FUNCTION_BLOCK XCBR (* Composite Function Block Type *)
  (* Standard: 61499-2 *)
  (* Version 0.0, 12/11/2023, Cheyan, Schneider Electric, template *)
  PACKAGE Main;
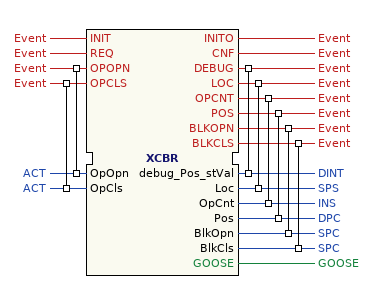
  EVENT_INPUT
    INIT; (* Initialization Request *)
    REQ; (* Normal Execution Request *)
    OPOPN WITH OpOpn;
    OPCLS WITH OpCls;
  END_EVENT
  EVENT_OUTPUT
    INITO; (* Initialization Confirm *)
    CNF; (* Execution Confirmation *)
    DEBUG WITH debug_Pos_stVal;
    LOC WITH Loc;
    OPCNT WITH OpCnt;
    POS WITH Pos;
    BLKOPN WITH BlkOpn;
    BLKCLS WITH BlkCls;
  END_EVENT
  VAR_INPUT
    OpOpn : ACT; (* Input event qualifier *)
    OpCls : ACT;
  END_VAR
  VAR_OUTPUT
    debug_Pos_stVal : DINT;
    Loc : SPS;
    OpCnt : INS;
    Pos : DPC;
    BlkOpn : SPC;
    BlkCls : SPC;
  END_VAR
  PLUGS
    GOOSE : GOOSE;
  END_PLUGS
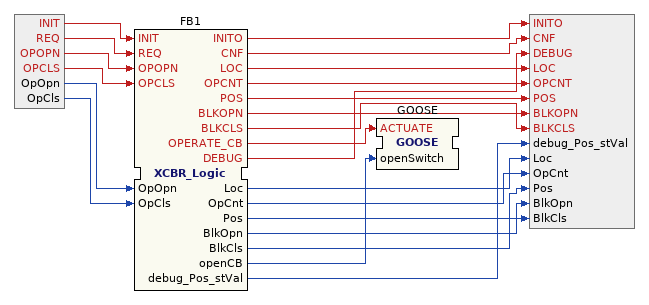
  FBS
    FB1 : XCBR_Logic;
  END_FBS
  EVENT_CONNECTIONS
    INIT TO FB1.INIT;
    REQ TO FB1.REQ;
    FB1.INITO TO INITO;
    FB1.CNF TO CNF;
    FB1.OPERATE_CB TO GOOSE.ACTUATE;
    FB1.DEBUG TO DEBUG;
    FB1.LOC TO LOC;
    FB1.OPCNT TO OPCNT;
    FB1.POS TO POS;
    FB1.BLKOPN TO BLKOPN;
    FB1.BLKCLS TO BLKCLS;
    OPOPN TO FB1.OPOPN;
    OPCLS TO FB1.OPCLS;
  END_CONNECTIONS
  DATA_CONNECTIONS
    FB1.openCB TO GOOSE.openSwitch;
    FB1.debug_Pos_stVal TO debug_Pos_stVal;
    FB1.Loc TO Loc;
    FB1.OpCnt TO OpCnt;
    FB1.Pos TO Pos;
    FB1.BlkOpn TO BlkOpn;
    FB1.BlkCls TO BlkCls;
    OpOpn TO FB1.OpOpn;
    OpCls TO FB1.OpCls;
  END_CONNECTIONS
END_FUNCTION_BLOCK
